{attribute 'linkalways'} 
{attribute 'no_explicit_call' := 'This FB is a CLASS and must be accessed using methods or properties'}
{attribute 'enable_dynamic_creation'}
FUNCTION_BLOCK _TOD EXTENDS DatatypeBase
VAR
	localData : TOD;
	activeData : REFERENCE TO TOD REF= localData;
END_VAR

PROPERTY PUBLIC Address : PVOID
GET
Address := ADR(activeData);
END_GET
END_PROPERTY

METHOD PUBLIC ClearReference
VAR_INPUT
END_VAR
activeData REF= localData;
END_METHOD

METHOD PUBLIC Clone : I_Datatype
VAR
    pClone : POINTER TO _TOD;
END_VAR
pClone := __NEW(_TOD(InitialValue := Value));
Clone := pClone^;
END_METHOD

METHOD FB_init : BOOL
VAR_INPUT
	bInitRetains : BOOL; // if TRUE, the retain variables are initialized (warm start / cold start)
	bInCopyCode : BOOL;  // if TRUE, the instance afterwards gets moved WORDo the copy code (online change)
	InitialValue : TOD;
END_VAR
localData := InitialValue;
END_METHOD

METHOD PUBLIC MakeReferenceTo
VAR_INPUT
	ReferenceTarget : REFERENCE TO TOD;
END_VAR
activeData REF= ReferenceTarget;
END_METHOD

PROPERTY PUBLIC Name : T_MAXSTRING
GET
Name := 'TOD';
END_GET
END_PROPERTY

METHOD PUBLIC SerializeWith
VAR_INPUT
	Serializer : I_Serializer;
END_VAR
Serializer.AddTod(activeData);
END_METHOD

PROPERTY PUBLIC Size : UDINT
GET
Size := SIZEOF(activeData);
END_GET
END_PROPERTY

METHOD TryDeserializeFrom : BOOL
VAR_INPUT
	Deserializer : I_Deserializer;
	Feedback : I_DeserializerFeedback;
END_VAR
TryDeserializeFrom := Deserializer.TryGetTod(activeData, Feedback);
END_METHOD

METHOD TryMakeReferenceTo : BOOL
VAR_INPUT
	Target : I_Datatype;
END_VAR
VAR
	pTargetData : POINTER TO TOD;
END_VAR
IF NOT (Target.Name = Name) THEN
	RETURN;
END_IF

pTargetData := Target.Address;
activeData REF= pTargetData^;
TryMakeReferenceTo := TRUE;
END_METHOD

PROPERTY PUBLIC Value : TOD
GET
Value := activeData;
END_GET
SET
activeData := Value;
END_SET
END_PROPERTY

END_FUNCTION_BLOCK

(* stored: Version 1.1.0.1, ProductVersion 3.1.4024.12
   POU _TOD: Id {5654ec3c-c489-05cb-386c-950edeff45ba}, SpecialFunc None
   Folder Constructor: Id {0243146b-7820-0c1d-095d-84ae9b933681}
   Property Address: Id {f3e72f4b-4242-0197-2b22-2a32537a8fca}
   Get Get: Id {3418d08b-4089-0ecc-3584-cf0c7db45f71}
   Method ClearReference: Id {ca20eed4-6f91-0058-183c-8aad877ee675}
   Method Clone: Id {d013eb03-a13c-0d90-0b85-cc900d1282f0}
   Method FB_init: Id {1fef93ef-d45c-0427-3731-9fe77acf6b60}
   Method MakeReferenceTo: Id {fb0d8c1e-56fa-06d9-2f31-c215702d405c}
   Property Name: Id {abc475e6-e67b-0508-06a2-e36c33316dfe}
   Get Get: Id {3bb2b9ad-4c13-0e64-0f86-3ee28d4ecd4f}
   Method SerializeWith: Id {693c27f2-6d9a-02f9-3c5c-f6e3b0c9c457}
   Property Size: Id {c29fbc59-a523-0abe-07ca-75c1dff30def}
   Get Get: Id {24a40110-e6cb-0779-1f26-0ca24781d22f}
   Method TryDeserializeFrom: Id {445dc623-9a0a-09be-0e61-d7fa9409560f}
   Method TryMakeReferenceTo: Id {e2368570-5e2d-032a-317d-afa5cd4a83ba}
   Property Value: Id {7a0fd7c5-2786-029a-39a1-259d5b5bf786}
   Get Get: Id {a6ad1565-34ad-0c76-2c9c-07a9df958985}
   Set Set: Id {6d6f0635-91e5-06e6-3b8b-040c3883e2fa} *)
